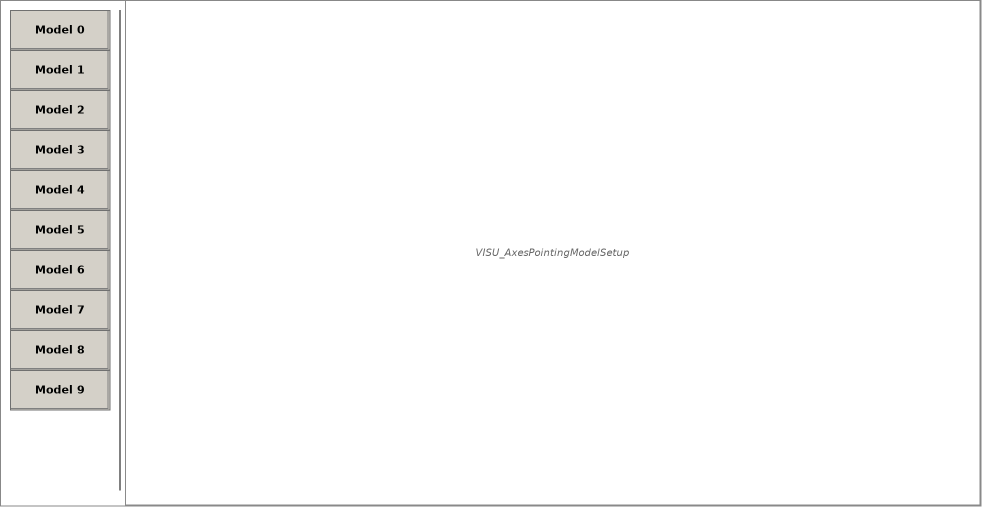
VISUALIZATION VISU_AxesPointingModelsSetup  // 982x507
VAR_IN_OUT
    ref : AxesPointingModelsSetup;
    widget : AxesPointingModelsSetupWidget;
END_VAR
    Button (10,10 100x40), "Model 0", pressed state: widget.activeModel = 0
        OnMouseClick: execute { widget.activeModel := 0; }
    Button (10,50 100x40), "Model 1", pressed state: widget.activeModel = 1
        OnMouseClick: execute { widget.activeModel := 1; }
    Button (10,90 100x40), "Model 2", pressed state: widget.activeModel = 2
        OnMouseClick: execute { widget.activeModel := 2; }
    Button (10,130 100x40), "Model 3", pressed state: widget.activeModel = 3
        OnMouseClick: execute { widget.activeModel := 3; }
    Button (10,170 100x40), "Model 4", pressed state: widget.activeModel = 4
        OnMouseClick: execute { widget.activeModel := 4; }
    Button (10,210 100x40), "Model 5", pressed state: widget.activeModel = 5
        OnMouseClick: execute { widget.activeModel := 5; }
    Button (10,250 100x40), "Model 6", pressed state: widget.activeModel = 6
        OnMouseClick: execute { widget.activeModel := 6; }
    Button (10,290 100x40), "Model 7", pressed state: widget.activeModel = 7
        OnMouseClick: execute { widget.activeModel := 7; }
    Button (10,330 100x40), "Model 8", pressed state: widget.activeModel = 8
        OnMouseClick: execute { widget.activeModel := 8; }
    Button (10,370 100x40), "Model 9", pressed state: widget.activeModel = 9
        OnMouseClick: execute { widget.activeModel := 9; }
    Frame (125,0 855x505), frame switch variable: widget.activeModel
        shows VISU_AxesPointingModelSetup(ref := ref.parts.model0, widget := widget.model0)
        shows VISU_AxesPointingModelSetup(ref := ref.parts.model1, widget := widget.model1)
        shows VISU_AxesPointingModelSetup(ref := ref.parts.model2, widget := widget.model2)
        shows VISU_AxesPointingModelSetup(ref := ref.parts.model3, widget := widget.model3)
        shows VISU_AxesPointingModelSetup(ref := ref.parts.model4, widget := widget.model4)
        shows VISU_AxesPointingModelSetup(ref := ref.parts.model5, widget := widget.model5)
        shows VISU_AxesPointingModelSetup(ref := ref.parts.model6, widget := widget.model6)
        shows VISU_AxesPointingModelSetup(ref := ref.parts.model7, widget := widget.model7)
        shows VISU_AxesPointingModelSetup(ref := ref.parts.model8, widget := widget.model8)
        shows VISU_AxesPointingModelSetup(ref := ref.parts.model9, widget := widget.model9)
    Line (120,490) (120,10)
END_VISUALIZATION

(* stored: Version 1.1.0.1, ProductVersion 3.1.4019.2
   Visu VISU_AxesPointingModelsSetup: Id {bba85ee3-6cc8-401c-806c-1e586a1135fb} *)
